Staubli VAL3: insert_dIn.pgx

public program insert_dIn(string x_sItem (dimensions=1), bool x_bActive (dimensions=1), dio x_dDio (dimensions=1))
begin
  // insert a new IO
  if isDefined(dInput[x_sItem])==false and ioStatus(x_dDio)>=0
    insert(dInput[x_sItem])
    dInput[x_sItem].bActive=x_bActive
    dInput[x_sItem].sID=x_sItem
    dInput[x_sItem].sName=x_sItem
    dioLink(dInput[x_sItem].dDio,x_dDio)
    dInput[x_sItem].bEnable=true
  endIf
end
